# B&R Automation Studio project Nitto (part 10)

#### FB_AxisCrtl_Home.st
```iecst
(********************************************************************
 * COPYRIGHT -- Microsoft
 ********************************************************************
 * Library: Bibliothek
 * Datei: FB_AxisCrtl_Home.st
 * Autor: awalz
 * Erstellt: 23. Juli 2014
 ********************************************************************
 * Implementierung der Library Bibliothek
 ********************************************************************)

(* TODO: Bitte Kommentar hier einfügen *)
FUNCTION_BLOCK FB_AxisCrtl_Home

(***************************************************************
        Control Sequence
***************************************************************)
(* status information is read before the step sequencer to attain a shorter reaction time *)
(************************ MC_READSTATUS *************************)
	MC_ReadStatus_0.Enable :=  NOT MC_ReadStatus_0.Error;
	MC_ReadStatus_0.Axis := AxisREF;
	MC_ReadStatus_0();
	BasicControl.AxisState.Disabled             := MC_ReadStatus_0.Disabled;
	BasicControl.AxisState.StandStill           := MC_ReadStatus_0.StandStill;
	BasicControl.AxisState.Stopping             := MC_ReadStatus_0.Stopping;
	BasicControl.AxisState.Homing               := MC_ReadStatus_0.Homing;
	BasicControl.AxisState.DiscreteMotion       := MC_ReadStatus_0.DiscreteMotion;
	BasicControl.AxisState.ContinuousMotion     := MC_ReadStatus_0.ContinuousMotion;
	BasicControl.AxisState.SynchronizedMotion   := MC_ReadStatus_0.SynchronizedMotion;
	BasicControl.AxisState.ErrorStop            := MC_ReadStatus_0.Errorstop;
	BasicControl.AxisState.Homed				:= BasicControl.Status.DriveStatus.HomingOk;
	(********************MC_BR_READDRIVESTATUS***********************)
	MC_BR_ReadDriveStatus_0.Enable := NOT(MC_BR_ReadDriveStatus_0.Error);
	MC_BR_ReadDriveStatus_0.Axis := AxisREF;
	MC_BR_ReadDriveStatus_0.AdrDriveStatus := ADR(BasicControl.Status.DriveStatus);
	MC_BR_ReadDriveStatus_0();

	(******************** MC_READACTUALPOSITION *********************)
	MC_ReadActualPosition_0.Enable := (NOT(MC_ReadActualPosition_0.Error));
	MC_ReadActualPosition_0.Axis := AxisREF;
	MC_ReadActualPosition_0();
	IF(MC_ReadActualPosition_0.Valid = TRUE)THEN
		BasicControl.Status.ActPosition := MC_ReadActualPosition_0.Position;
	END_IF

	(******************** MC_READACTUALVELOCITY *********************)
	MC_ReadActualVelocity_0.Enable := (NOT(MC_ReadActualVelocity_0.Error));
	MC_ReadActualVelocity_0.Axis := AxisREF;
	MC_ReadActualVelocity_0();
	IF(MC_ReadActualVelocity_0.Valid = TRUE)THEN
		BasicControl.Status.ActVelocity := MC_ReadActualVelocity_0.Velocity;
	END_IF
	(*********************+*Parameter schreiben**********************)
	MC_MoveVelocity_0.Acceleration  := ruck;
	MC_MoveVelocity_0.Deceleration  := ruck;
	MC_ReadStatus_0();
	(************************ MC_READAXISERROR **********************)
	MC_ReadAxisError_0.Enable := NOT(MC_ReadAxisError_0.Error);
	MC_ReadAxisError_0.Axis := AxisREF;
	MC_ReadAxisError_0.DataAddress := ADR(BasicControl.Status.ErrorText);
	MC_ReadAxisError_0.DataLength := SIZEOF(BasicControl.Status.ErrorText);
	MC_ReadAxisError_0.DataObjectName := 'acp10etxde';
	MC_ReadAxisError_0();

	MC_refSwitchConfig_0.Axis := AxisREF;
	MC_refSwitchConfig_0();

	(* central monitoring OF stop command attains a shorter reaction TIME in CASE OF emergency stop *)
	(******************CHECK FOR STOP COMMAND************************)
	(*IF (BasicControl.Command.Stop = TRUE) THEN*)
	IF cmd = CONST.AXIS.STOP THEN
		IF ((AxisStep >= STATE_READY) AND (AxisStep < STATE_ERROR)) THEN
			(* reset all FB execute inputs we use *)
			MC_Home_0.Execute := 0;
			MC_Stop_0.Execute := 0;
			MC_MoveAbsolute_0.Execute := 0;
			MC_MoveAdditive_0.Execute := 0;
			MC_MoveVelocity_0.Execute := 0;
			MC_ReadAxisError_0.Acknowledge := 0;
			MC_Reset_0.Execute := 0;

			(* reset user commands *)
			BasicControl.Command.Stop := 0;
			BasicControl.Command.Home := 0;
			BasicControl.Command.MoveJogPos := 0;
			BasicControl.Command.MoveJogNeg := 0;
			BasicControl.Command.MoveVelocity := 0;
			BasicControl.Command.MoveAbsolute := 0;
			BasicControl.Command.MoveAdditive := 0;
			AxisStep := STATE_STOP;
		END_IF
	END_IF

//////////////////////////////////////////////////////////////////////////
(*	IF AxisHandle[tempIndex].AxisState.Stopping THEN
	    IF (AxisHandle[tempIndex].Status.ActVelocity = 0.0) THEN
			AxisIf.Status.isMoving 						:= FALSE;
			AllDrives.Status.stopActive					:= FALSE;
		ELSE
			AxisIf.Status.isMoving 						:= TRUE;
		END_IF
	ELSIF (NOT ( AxisHandle[tempIndex].AxisState.DiscreteMotion OR
	             AxisHandle[tempIndex].AxisState.ContinuousMotion)) THEN
		AxisIf.Status.isMoving 							:= FALSE;
		AllDrives.Status.stopActive						:= FALSE;
	ELSE
		AxisIf.Status.isMoving 							:= TRUE;
	END_IF*)
////////////////////////////////////////////////////////////////////////////
	(**************** CHECK FOR GENERAL AXIS ERROR ******************)
(*	IF ((MC_ReadAxisError_0.AxisErrorID <> 0) AND (MC_ReadAxisError_0.Valid)) THEN
		AxisStep := STATE_ERROR_AXIS;
		(***************** CHECK IF POWER SHOULD BE OFF *******************)
(*	ELSIF ((NOT BasicControl.Command.Power) AND (MC_ReadAxisError_0.Valid)) THEN
		IF ((MC_ReadStatus_0.Errorstop) AND (MC_ReadStatus_0.Valid )) THEN
			AxisStep := STATE_ERROR_RESET;
		ELSE
			AxisStep := STATE_WAIT;
		END_IF
	END_IF*)

	CASE AxisStep OF

//		******************* WAIT ************************
		STATE_WAIT:  (* STATE: Wait *)
			AxisStep := STATE_QUIT;
//			(*IF (BasicControl.Command.Power = TRUE) THEN*)
//			IF cmd = CONST.AXIS.POWER_ON THEN
//				cmdtmp := cmd;
//				AxisStep := STATE_POWER_ON;
//			ELSIF cmd = CONST.AXIS.VAXIS_ON THEN
//				cmdtmp := cmd;
//				AxisStep := STATE_VAXIS_ON;
//			ELSIF cmd = CONST.AXIS.POWER_OFF THEN
//				cmdtmp := cmd;
//				AxisStep := STATE_POWER_OFF;
//			ELSE
//				MC_Power_0.Enable := FALSE;
//			END_IF
//
//			(* reset all FB execute inputs we use *)
//			MC_Home_0.Execute := FALSE;
//			MC_Stop_0.Execute := FALSE;
//			MC_MoveAbsolute_0.Execute := FALSE;
//			MC_MoveAdditive_0.Execute := FALSE;
//			MC_MoveVelocity_0.Execute := FALSE;
//			MC_ReadAxisError_0.Acknowledge := FALSE;
//			MC_Reset_0.Execute := FALSE;
//			(* reset user commands *)
//			BasicControl.Command.Stop := FALSE;
//			BasicControl.Command.Home := FALSE;
//			BasicControl.Command.MoveJogPos := FALSE;
//			BasicControl.Command.MoveJogNeg := FALSE;
//			BasicControl.Command.MoveVelocity := FALSE;
//			BasicControl.Command.MoveAbsolute := FALSE;
//			BasicControl.Command.MoveAdditive := FALSE;
//
//			BasicControl.Status.ErrorID := 0;
//		(********************Virtuelle Achse einschalten****)
		STATE_VAXIS_ON:

			IF MC_BR_ReadDriveStatus_0.Valid THEN
				cmdtmp := cmd;
				AxisStep := STATE_QUIT;
			END_IF
		(******************** POWER ON **********************)
		STATE_POWER_ON:  (* STATE: Power on *)
			(*MC_Power_0.Enable := TRUE;*)
			IF (*BasicControl.Status.DriveStatus.ControllerReady AND *) BasicControl.Status.DriveStatus.NetworkInit AND
			cmd = CONST.AXIS.POWER_ON AND NOT MC_Power_0.Status AND NOT MC_Power_0.Error THEN
				MC_Power_0.Enable := TRUE; (*erster Anlauf*)
			ELSIF MC_Power_0.Error AND cmd = CONST.AXIS.POWER_ON THEN
					MC_Power_0.Enable := FALSE ;(* if a power error occured go to error state *)
					cmdtmp := cmd;
					AxisStep := STATE_ERROR_RESET;
			ELSIF 	MC_Power_0.Status AND NOT MC_Power_0.Error THEN
					cmdtmp := cmd;
					AxisStep := STATE_QUIT;
			ELSIF MC_ReadStatus_0.Errorstop AND cmdtmp <> cmd THEN
					BasicControl.Status.ErrorID := MC_Power_0.ErrorID;
					AxisStep := STATE_ERROR;
			END_IF
		(******************** POWER OFF **********************)
		STATE_POWER_OFF:  (* STATE: Power on *)
			MC_Power_0.Enable := FALSE;
			IF NOT MC_Power_0.Status THEN
				cmdtmp := cmd;
				AxisStep := STATE_QUIT;
			END_IF
			(* if a power error occured go to error state *)
			IF MC_Power_0.Error  THEN
				BasicControl.Status.ErrorID := MC_Power_0.ErrorID;
				AxisStep := STATE_ERROR;
			ELSIF MC_ReadStatus_0.Errorstop AND cmdtmp <> cmd THEN
				AxisStep := STATE_ERROR_RESET;
			END_IF
		(******************** READY **********************)
		STATE_READY:  (* STATE: Waiting for commands *)
			IF cmd <> CONST.AXIS.NOACTION THEN
					busy := TRUE;
					cmdtmp:= cmd;
					IF cmd = CONST.AXIS.RESET THEN
						AxisStep := STATE_ERROR_RESET;
					ELSIF cmd = CONST.AXIS.STOP THEN
						MC_Stop_0( Execute := TRUE, Deceleration := verzoegerung);
						AxisStep := STATE_STOP;
					ELSIF cmd = CONST.AXIS.JOG_NEG THEN
						MC_MoveVelocity_0(Execute := TRUE, Velocity := 16666*velocity,Direction := mcNEGATIVE_DIR,
								Acceleration  := BasicControl.Parameter.Acceleration, Deceleration := BasicControl.Parameter.Deceleration);
						AxisStep := STATE_JOG_NEGATIVE;
					ELSIF cmd = CONST.AXIS.JOG_POS THEN
						MC_MoveVelocity_0(Execute := TRUE, Velocity := 16666*velocity,Direction := mcPOSITIVE_DIR,
									Acceleration  := BasicControl.Parameter.Acceleration, Deceleration := BasicControl.Parameter.Deceleration);
						AxisStep := STATE_JOG_POSITIVE;
					ELSIF cmd = CONST.AXIS.SETPOS THEN
						MC_MoveAbsolute_0(Execute := TRUE, Position := position, Velocity := 16666*velocity, Direction := mcPOSITIVE_DIR,
								Acceleration  := BasicControl.Parameter.Acceleration, Deceleration := BasicControl.Parameter.Deceleration);
						AxisStep := STATE_MOVE_ABSOLUTE; (*STATE_MOVE_ADDITIVE*)(*STATE_MOVE_ABSOLUTE;*)
					ELSIF  cmd = CONST.AXIS.CALIBR THEN
						MC_Home_0(Execute := TRUE, Position := BasicControl.Parameter.HomePosition, HomingMode := BasicControl.Parameter.HomeMode);
						AxisStep := STATE_HOME;
					ELSIF cmd = CONST.AXIS.MOVE_VELOCITY THEN
							MC_MoveVelocity_0(Execute := TRUE, Velocity := 16666*velocity,Direction := mcPOSITIVE_DIR);
						AxisStep := STATE_MOVE_VELOCITY;
					ELSIF   cmd = CONST.AXIS.POWER_OFF THEN
						AxisStep := STATE_POWER_OFF;
					ELSIF   cmd = CONST.AXIS.POWER_ON THEN
						AxisStep := STATE_POWER_ON;
					END_IF
			(*ELSE
				busy := FALSE;*)
			END_IF
		(******************** HOME **********************)
		STATE_HOME:  (* STATE: start homing process *)
//			IF cmd = CONST.AXIS.CALIBR AND NOT MC_Home_0.Done THEN
//				MC_Home_0.Execute := TRUE;
			IF MC_Home_0.Done AND cmd = CONST.AXIS.CALIBR THEN
				MC_Home_0.Execute := FALSE;
				BasicControl.AxisState.Homed := TRUE;
				cmdtmp := cmd;
				busy := FALSE;
				AxisStep := STATE_QUIT;
			ELSIF cmd <> CONST.AXIS.CALIBR THEN
				MC_Home_0.Execute := FALSE;
				MC_Stop_0( Execute := TRUE, Deceleration := verzoegerung);
				AxisStep := STATE_STOP;
			END_IF
			(* if a homing error occured go to error state *)
			IF MC_Home_0.Error  OR MC_ReadStatus_0.Errorstop THEN
				MC_Home_0.Execute := FALSE;
				BasicControl.Status.ErrorID := MC_Home_0.ErrorID;
				AxisStep := STATE_ERROR;
			END_IF

		(***********************HALT_MOVEMENT***************************)
		STATE_HALT:   (* STATE: Halt movement *)
			MC_Halt_0.Deceleration := BasicControl.Parameter.Deceleration;
			MC_Halt_0.Execute := TRUE;
			IF MC_Halt_0.Done OR MC_Halt_0.CommandAborted THEN
				MC_Halt_0.Execute := FALSE;
				cmdtmp := cmd;
				busy := FALSE;
				AxisStep := STATE_QUIT;
			ELSIF cmd = CONST.AXIS.STOP THEN
				MC_Halt_0.Execute := FALSE;
				MC_Stop_0( Execute := TRUE, Deceleration := verzoegerung);
				AxisStep := STATE_STOP;
			END_IF
			(* check if error occured *)
			IF MC_Halt_0.Error OR  MC_ReadStatus_0.Errorstop THEN
				BasicControl.Status.ErrorID := MC_Halt_0.ErrorID;
				MC_Halt_0.Execute := FALSE;
				AxisStep := STATE_ERROR;
			END_IF

		(*********************** STOP MOVEMENT *************************)
		STATE_STOP: //9  (* STATE: Stop movement *)
			(* if axis is stopped go to ready state *)
			MC_Stop_0.Execute := TRUE;
			IF MC_Stop_0.Done OR MC_ReadStatus_0.StandStill THEN
				MC_Stop_0.Execute := FALSE;
				cmdtmp := cmd;
				AxisStep := STATE_QUIT;
			ELSIF MC_ReadStatus_0.Disabled THEN
				MC_Stop_0.Execute := FALSE;
				cmdtmp := cmd;
				AxisStep := STATE_QUIT;
			END_IF
			(* check if error occured *)
			IF MC_Stop_0.Error OR MC_ReadStatus_0.Errorstop THEN
				BasicControl.Status.ErrorID := MC_Stop_0.ErrorID;
				MC_Stop_0.Execute := FALSE;
				AxisStep := STATE_ERROR;
			END_IF

		(******************** START JOG MOVEMENT POSITVE **********************)
		STATE_JOG_POSITIVE:  (* STATE: Start jog movement in positive direction *)
			IF cmd <> CONST.AXIS.JOG_POS AND cmd <> CONST.AXIS.STOP THEN
				cmdtmp := cmd;
				MC_MoveVelocity_0.Execute := FALSE;
				AxisStep := STATE_HALT;
			ELSIF cmd = CONST.AXIS.STOP THEN
				MC_MoveVelocity_0.Execute := FALSE;
				MC_Stop_0( Execute := TRUE, Deceleration := verzoegerung);
				AxisStep := STATE_STOP;
			END_IF
			(* check if error occured *)
			IF MC_MoveVelocity_0.Error OR MC_ReadStatus_0.Errorstop  THEN
				BasicControl.Status.ErrorID := MC_MoveVelocity_0.ErrorID;
				MC_MoveVelocity_0.Execute := FALSE;
				AxisStep := STATE_ERROR;
			END_IF

		(******************** START JOG MOVEMENT NEGATIVE **********************)
		STATE_JOG_NEGATIVE:  (* STATE: Start jog movement in negative direction *)

			IF cmd <> CONST.AXIS.JOG_NEG AND  cmd <> CONST.AXIS.STOP THEN
				MC_MoveVelocity_0.Execute := FALSE;
				cmdtmp := cmd;
				AxisStep := STATE_HALT;
			ELSIF cmd = CONST.AXIS.STOP THEN
				MC_MoveVelocity_0.Execute := FALSE;
				MC_Stop_0( Execute := TRUE, Deceleration := verzoegerung);
				AxisStep := STATE_STOP;
			END_IF
			(* check if error occured *)
			IF MC_MoveVelocity_0.Error OR MC_ReadStatus_0.Errorstop THEN
				BasicControl.Status.ErrorID := MC_MoveVelocity_0.ErrorID;
				MC_MoveVelocity_0.Execute := FALSE;
				AxisStep := STATE_ERROR;
			END_IF

		(******************** START ABSOLUTE MOVEMENT **********************)
		STATE_MOVE_ABSOLUTE:  (* STATE: Start absolute movement *)
			(* check if commanded position is reached *)
			IF cmd <> CONST.AXIS.SETPOS AND cmd <> CONST.AXIS.STOP  THEN
				MC_MoveAbsolute_0.Execute := FALSE;
				cmdtmp := cmd;
				AxisStep := STATE_HALT;
			ELSIF MC_MoveAbsolute_0.Done THEN
				MC_MoveAbsolute_0.Execute := FALSE;
				cmdtmp := cmd;
				AxisStep := STATE_QUIT;
			ELSIF cmd = CONST.AXIS.STOP THEN
				MC_MoveAbsolute_0.Execute := FALSE;
				MC_Stop_0.Deceleration := verzoegerung;
				MC_Stop_0.Execute := TRUE;
				AxisStep := STATE_STOP;
			END_IF
			(* check if error occured *)
			IF MC_MoveAbsolute_0.Error OR MC_ReadStatus_0.Errorstop THEN
				BasicControl.Status.ErrorID := MC_MoveAbsolute_0.ErrorID;
				MC_MoveAbsolute_0.Execute := TRUE;
				AxisStep := STATE_ERROR;
			END_IF

		(******************** START ADDITIVE MOVEMENT **********************)
		STATE_MOVE_ADDITIVE:  (* STATE: Start additive movement *)
			(*	MC_MoveAdditive_0.Distance      := BasicControl.Parameter.Distance;
			MC_MoveAdditive_0.Velocity      := BasicControl.Parameter.Velocity;
			MC_MoveAdditive_0.Execute := TRUE;*)
			MC_MoveAdditive_0.Acceleration  := BasicControl.Parameter.Acceleration;
			MC_MoveAdditive_0.Deceleration  := BasicControl.Parameter.Deceleration;

			(* check if commanded distance is reached *)
			IF cmd <> CONST.AXIS.SETPOS AND cmd <> CONST.AXIS.STOP THEN
				MC_MoveAdditive_0.Execute := FALSE;
				cmdtmp := cmd;
				AxisStep := STATE_HALT;
			ELSIF MC_MoveAdditive_0.Done  THEN
				MC_MoveAdditive_0.Execute := FALSE;
				cmdtmp := cmd;
				AxisStep := STATE_QUIT;
			ELSIF cmd = CONST.AXIS.STOP THEN
				MC_MoveAdditive_0.Execute := FALSE;
				MC_Stop_0( Execute := TRUE, Deceleration := verzoegerung);
				AxisStep := STATE_STOP;
			END_IF
			(* check if error occured *)
			IF MC_MoveAdditive_0.Error OR  MC_ReadStatus_0.Errorstop THEN
				BasicControl.Status.ErrorID := MC_MoveAdditive_0.ErrorID;
				MC_MoveAdditive_0.Execute := FALSE;
				AxisStep := STATE_ERROR;
			END_IF

		(******************** START VELOCITY MOVEMENT **********************)
		STATE_MOVE_VELOCITY:  (* STATE: Start velocity movement *)
					(* check if commanded velocity is reached *)
			IF cmd <>  CONST.AXIS.MOVE_VELOCITY AND  cmd <> CONST.AXIS.STOP THEN
				MC_MoveVelocity_0.Execute := FALSE;
				cmdtmp := cmd;
				AxisStep := STATE_HALT;
			ELSIF MC_MoveVelocity_0.InVelocity THEN
				MC_MoveVelocity_0.Execute := FALSE;
				cmdtmp := cmd;
				AxisStep := STATE_QUIT;
			ELSIF cmd = CONST.AXIS.STOP THEN
				MC_MoveVelocity_0.Execute := FALSE;
				MC_Stop_0( Execute := TRUE, Deceleration := verzoegerung);
				AxisStep := STATE_STOP;
			END_IF
			(* check if error occured *)
			IF MC_MoveVelocity_0.Error OR MC_ReadStatus_0.Errorstop THEN
				BasicControl.Status.ErrorID := MC_MoveVelocity_0.ErrorID;
				MC_MoveVelocity_0.Execute := FALSE;
				AxisStep := STATE_ERROR;
			END_IF

		(******************** FB-ERROR OCCURED *************************)
		STATE_ERROR:  (* STATE: Error *)
			(* check if FB indicates an axis error *)
			IF (MC_ReadAxisError_0.AxisErrorCount<>0) THEN
				AxisStep := STATE_ERROR_AXIS;
			ELSE
				IF (BasicControl.Command.ErrorAcknowledge = TRUE) THEN
					BasicControl.Command.ErrorAcknowledge := FALSE;
					BasicControl.Status.ErrorID := 0;
					(* reset axis if it is in axis state ErrorStop *)
					IF MC_ReadStatus_0.Errorstop AND MC_ReadStatus_0.Valid  THEN
						AxisStep := STATE_ERROR_RESET;
					ELSE
						cmdtmp := cmd;
						AxisStep := STATE_QUIT;
					END_IF
				END_IF
			END_IF

		(******************** AXIS-ERROR OCCURED *************************)
		STATE_ERROR_AXIS:  (* STATE: Axis Error *)
			IF (MC_ReadAxisError_0.Valid) THEN
			err.set := TRUE;
			err.text := MC_ReadAxisError_0.DataObjectName;
			err.id :=  UINT_TO_DINT  (MC_ReadAxisError_0.AxisErrorID) ;
				IF (MC_ReadAxisError_0.AxisErrorID <> 0) THEN
					BasicControl.Status.ErrorID := MC_ReadAxisError_0.AxisErrorID;
				END_IF
				MC_ReadAxisError_0.Acknowledge := FALSE;
			(*	IF (BasicControl.Command.ErrorAcknowledge) THEN
					BasicControl.Command.ErrorAcknowledge := FALSE;
					(* acknowledge axis error *)
				IF cmd = CONST.AXIS.RESET THEN
					IF (MC_ReadAxisError_0.AxisErrorID <> 0) THEN
						MC_ReadAxisError_0.Acknowledge := TRUE;
						AxisStep := STATE_ERROR_RESET;
					END_IF
				END_IF
				IF (MC_ReadAxisError_0.AxisErrorCount = 0) THEN
					(* reset axis if it is in axis state ErrorStop *)
					BasicControl.Status.ErrorID := 0;
					IF ((MC_ReadStatus_0.Errorstop ) AND (MC_ReadStatus_0.Valid)) THEN
						AxisStep := STATE_ERROR_RESET;
					ELSE
						(*AxisStep := STATE_WAIT;*)
						cmdtmp := cmd;
						AxisStep := STATE_QUIT;
					END_IF
				ELSIF NOT MC_ReadAxisError_0.Error THEN
						cmdtmp := cmd;
							AxisStep := STATE_QUIT;
				END_IF
			ELSE
				AxisStep := STATE_WAIT; (* kein Fehler liegt vor*)
			END_IF

		(******************** RESET DONE *************************)
		STATE_ERROR_RESET:  (* STATE: Wait for reset done *)
			MC_Reset_0.Execute := TRUE;
			(* reset MC_Power.Enable if this FB is in Error*)
			IF (MC_Power_0.Error) THEN
				MC_Power_0.Enable := FALSE;
			END_IF
			IF(MC_Reset_0.Done)THEN
				MC_Reset_0.Execute := FALSE;
				(*AxisStep := STATE_WAIT;*)
				cmdtmp := cmd;
				(*cmd := CONST.AXIS.NOACTION;*)
				AxisStep := STATE_QUIT;
			ELSIF(MC_Reset_0.Error) THEN
				MC_Reset_0.Execute := FALSE;
				AxisStep := STATE_ERROR;
			END_IF
			(******************** SEQUENCE END *************************)
		STATE_QUIT:
		(*IF cmd = CONST.CUTTINGUNIT.CMDs.ABORT THEN
			busy := TRUE;
			state := ST_ABORT;
		ELSE*)
			busy := FALSE;
			IF cmd = cmdtmp THEN
				busy := FALSE;
				cmd := CONST.AXIS.NOACTION;
				AxisStep := STATE_READY;
			ELSIF cmd <> CONST.AXIS.NOACTION THEN
				busy := FALSE;
				AxisStep := STATE_READY;
			(*ELSIF cmd = CONST.AXIS.POWER_OFF THEN
				cmdtmp := cmd;
				AxisStep := STATE_POWER_OFF;*)
			(*ELSIF cmd = CONST.AXIS.POWER_ON THEN
				cmdtmp := cmd;
				AxisStep := STATE_POWER_ON;*)

			END_IF

	END_CASE

(***************************************************************
        FUNCTION Block Calls
***************************************************************)

(************************** MC_POWER ****************************)
	MC_Power_0.Axis := AxisREF;  (* pointer to axis *)
	MC_Power_0();

	(************************** MC_HOME *****************************)
	MC_Home_0.Axis := AxisREF;
	MC_Home_0();

	(********************** MC_MOVEABSOLUTE *************************)
	MC_MoveAbsolute_0.Axis := AxisREF;
	MC_MoveAbsolute_0();

	(********************** MC_MOVEADDITIVE *************************)
	MC_MoveAdditive_0.Axis := AxisREF;
	MC_MoveAdditive_0();

	(********************** MC_MOVEVELOCITY *************************)
	MC_MoveVelocity_0.Axis := AxisREF;
	MC_MoveVelocity_0();

	(************************** MC_STOP *****************************)
	MC_Stop_0.Axis := AxisREF;
	MC_Stop_0();

	(***************************MC_HALT******************************)
	MC_Halt_0.Axis := AxisREF;
	MC_Halt_0();

	(************************** MC_RESET ****************************)
	MC_Reset_0.Axis := AxisREF;
	MC_Reset_0();
END_FUNCTION_BLOCK
```

#### FB_AxisState.st
```iecst
(********************************************************************
 * COPYRIGHT -- Microsoft
 ********************************************************************
 * Library: Bibliothek
 * Datei: FB_AxisState.st
 * Autor: awalz
 * Erstellt: 26. August 2014
 ********************************************************************
 * Implementierung der Library Bibliothek
 ********************************************************************)

(* TODO: Bitte Kommentar hier einfügen *)
FUNCTION_BLOCK FB_AxisState
//		Error:				INT:=1;
//		Errorstop:			INT:=2;
//		Disabled:			INT:=3;
//		Stopping:			INT:=4;
//		StandStill:			INT:=5;
//		DiscreteMotion:		INT:=6;
//		ContinuousMotion: 	INT:=7;
//		SynchronizedMotion:	INT:=8;
//		Homing:				INT:=9;
	stati[CONST.Error] := readstatus.Error;
	stati[CONST.Errorstop] :=	readstatus.Errorstop;
	stati[CONST.Disabled] :=	readstatus.Disabled;
	stati[3] :=	readstatus.Stopping;
	stati[4] := readstatus.StandStill;
	stati[5] := readstatus.DiscreteMotion;
	stati[6] :=	readstatus.ContinuousMotion;
	stati[7] :=	readstatus.SynchronizedMotion;
//	CONST.texts[CONST.Error] := stati[0];
//
//
//		readstatus.SynchronizedMotion
END_FUNCTION_BLOCK
```

#### FB_AxisCtrl_GridFeeder.st
```iecst
(********************************************************************
 * COPYRIGHT -- Microsoft
 ********************************************************************
 * Library: Bibliothek
 * Datei: FB_AxisCtrl.st
 * Autor: awalz
 * Erstellt: 23. Juli 2014
 ********************************************************************
 * Implementierung der Library Bibliothek
 ********************************************************************)

(* TODO: Bitte Kommentar hier einfügen *)
FUNCTION_BLOCK FB_AxisCtrl_GridFeeder

(***************************************************************
        Control Sequence
***************************************************************)
(* status information is read before the step sequencer to attain a shorter reaction time *)
(************************ MC_READSTATUS *************************)
	MC_ReadStatus_0.Enable :=  NOT MC_ReadStatus_0.Error;
	MC_ReadStatus_0.Axis := AxisREF;
	MC_ReadStatus_0();
	BasicControl.AxisState.Disabled             := MC_ReadStatus_0.Disabled;
	BasicControl.AxisState.StandStill           := MC_ReadStatus_0.StandStill;
	BasicControl.AxisState.Stopping             := MC_ReadStatus_0.Stopping;
	BasicControl.AxisState.Homing               := MC_ReadStatus_0.Homing;
	BasicControl.AxisState.DiscreteMotion       := MC_ReadStatus_0.DiscreteMotion;
	BasicControl.AxisState.ContinuousMotion     := MC_ReadStatus_0.ContinuousMotion;
	BasicControl.AxisState.SynchronizedMotion   := MC_ReadStatus_0.SynchronizedMotion;
	BasicControl.AxisState.ErrorStop            := MC_ReadStatus_0.Errorstop;

	(********************MC_BR_READDRIVESTATUS***********************)
	MC_BR_ReadDriveStatus_0.Enable := NOT(MC_BR_ReadDriveStatus_0.Error);
	MC_BR_ReadDriveStatus_0.Axis := AxisREF;
	MC_BR_ReadDriveStatus_0.AdrDriveStatus := ADR(BasicControl.Status.DriveStatus);
	MC_BR_ReadDriveStatus_0();

	(******************** MC_READACTUALPOSITION *********************)
	MC_ReadActualPosition_0.Enable := (NOT(MC_ReadActualPosition_0.Error));
	MC_ReadActualPosition_0.Axis := AxisREF;
	MC_ReadActualPosition_0();
	IF(MC_ReadActualPosition_0.Valid = TRUE)THEN
		BasicControl.Status.ActPosition := MC_ReadActualPosition_0.Position;
	END_IF

	(******************** MC_READACTUALVELOCITY *********************)
	MC_ReadActualVelocity_0.Enable := (NOT(MC_ReadActualVelocity_0.Error));
	MC_ReadActualVelocity_0.Axis := AxisREF;
	MC_ReadActualVelocity_0();
	IF(MC_ReadActualVelocity_0.Valid = TRUE)THEN
		BasicControl.Status.ActVelocity := MC_ReadActualVelocity_0.Velocity;
	END_IF
	(*********************+*Parameter schreiben**********************)
	MC_MoveVelocity_0.Acceleration  := ruck;
	MC_MoveVelocity_0.Deceleration  := ruck;
	MC_ReadStatus_0();
	(************************ MC_READAXISERROR **********************)
	MC_ReadAxisError_0.Enable := NOT(MC_ReadAxisError_0.Error);
	MC_ReadAxisError_0.Axis := AxisREF;
	MC_ReadAxisError_0.DataAddress := ADR(BasicControl.Status.ErrorText);
	MC_ReadAxisError_0.DataLength := SIZEOF(BasicControl.Status.ErrorText);
	MC_ReadAxisError_0.DataObjectName := 'acp10etxde';
	MC_ReadAxisError_0();
	(* central monitoring OF stop command attains a shorter reaction TIME in CASE OF emergency stop *)
	(******************CHECK FOR STOP COMMAND************************)
	(*IF (BasicControl.Command.Stop = TRUE) THEN*)
	//	IF cmd = CONST.AXIS.STOP THEN //12.03.15
	//		busy := TRUE;
	//		IF ((AxisStep >= STATE_READY) AND (AxisStep < STATE_ERROR)) THEN
	//			(* reset all FB execute inputs we use *)
	//			MC_Home_0.Execute := 0;
	//			MC_Stop_0.Execute := 0;
	//			MC_MoveAbsolute_0.Execute := 0;
	//			MC_MoveAdditive_0.Execute := 0;
	//			MC_MoveVelocity_0.Execute := 0;
	//			MC_ReadAxisError_0.Acknowledge := 0;
	//			MC_Reset_0.Execute := 0;
	//
	//			(* reset user commands *)
	//			BasicControl.Command.Stop := 0;
	//			BasicControl.Command.Home := 0;
	//			BasicControl.Command.MoveJogPos := 0;
	//			BasicControl.Command.MoveJogNeg := 0;
	//			BasicControl.Command.MoveVelocity := 0;
	//			BasicControl.Command.MoveAbsolute := 0;
	//			BasicControl.Command.MoveAdditive := 0;
	//			MC_Stop_0( Execute := TRUE, Deceleration := verzoegerung);
	//			AxisStep := STATE_STOP;
	//		END_IF
	//	END_IF
	//
	////////////////////////////////////////////////////////////////////////////
	//(*	IF AxisHandle[tempIndex].AxisState.Stopping THEN
	//	    IF (AxisHandle[tempIndex].Status.ActVelocity = 0.0) THEN
	//			AxisIf.Status.isMoving 						:= FALSE;
	//			AllDrives.Status.stopActive					:= FALSE;
	//		ELSE
	//			AxisIf.Status.isMoving 						:= TRUE;
	//		END_IF
	//	ELSIF (NOT ( AxisHandle[tempIndex].AxisState.DiscreteMotion OR
	//	             AxisHandle[tempIndex].AxisState.ContinuousMotion)) THEN
	//		AxisIf.Status.isMoving 							:= FALSE;
	//		AllDrives.Status.stopActive						:= FALSE;
	//	ELSE
	//		AxisIf.Status.isMoving 							:= TRUE;
	//	END_IF*)
	//////////////////////////////////////////////////////////////////////////////
	//	(**************** CHECK FOR GENERAL AXIS ERROR ******************)
	//(*	IF ((MC_ReadAxisError_0.AxisErrorID <> 0) AND (MC_ReadAxisError_0.Valid)) THEN
	//		AxisStep := STATE_ERROR_AXIS;
	//		(***************** CHECK IF POWER SHOULD BE OFF *******************)
	//(*	ELSIF ((NOT BasicControl.Command.Power) AND (MC_ReadAxisError_0.Valid)) THEN
	//		IF ((MC_ReadStatus_0.Errorstop) AND (MC_ReadStatus_0.Valid )) THEN
	//			AxisStep := STATE_ERROR_RESET;
	//		ELSE
	//			AxisStep := STATE_WAIT;
	//		END_IF
	//	END_IF*)

	CASE AxisStep OF

		//		******************* WAIT ************************
		STATE_WAIT:  (* STATE: Wait *)
			AxisStep := STATE_QUIT;
		//			(*IF (BasicControl.Command.Power = TRUE) THEN*)
		//			IF cmd = CONST.AXIS.POWER_ON THEN
		//				cmdtmp := cmd;
		//				AxisStep := STATE_POWER_ON;
		//			ELSIF cmd = CONST.AXIS.VAXIS_ON THEN
		//				cmdtmp := cmd;
		//				AxisStep := STATE_VAXIS_ON;
		//			ELSIF cmd = CONST.AXIS.POWER_OFF THEN
		//				cmdtmp := cmd;
		//				AxisStep := STATE_POWER_OFF;
		//			ELSE
		//				MC_Power_0.Enable := FALSE;
		//			END_IF
		//
		//			(* reset all FB execute inputs we use *)
		//			MC_Home_0.Execute := FALSE;
		//			MC_Stop_0.Execute := FALSE;
		//			MC_MoveAbsolute_0.Execute := FALSE;
		//			MC_MoveAdditive_0.Execute := FALSE;
		//			MC_MoveVelocity_0.Execute := FALSE;
		//			MC_ReadAxisError_0.Acknowledge := FALSE;
		//			MC_Reset_0.Execute := FALSE;
		//			(* reset user commands *)
		//			BasicControl.Command.Stop := FALSE;
		//			BasicControl.Command.Home := FALSE;
		//			BasicControl.Command.MoveJogPos := FALSE;
		//			BasicControl.Command.MoveJogNeg := FALSE;
		//			BasicControl.Command.MoveVelocity := FALSE;
		//			BasicControl.Command.MoveAbsolute := FALSE;
		//			BasicControl.Command.MoveAdditive := FALSE;
		//
		//			BasicControl.Status.ErrorID := 0;
		//		(********************Virtuelle Achse einschalten****)
		STATE_VAXIS_ON:

			IF MC_BR_ReadDriveStatus_0.Valid THEN
				cmdtmp := cmd;
				AxisStep := STATE_QUIT;
			END_IF
		(******************** POWER ON **********************)
		STATE_POWER_ON:  (* STATE: Power on *)
			(*MC_Power_0.Enable := TRUE;*)
			IF BasicControl.Status.DriveStatus.ControllerReady AND	cmd = CONST.AXIS.POWER_ON
				AND NOT MC_Power_0.Status AND NOT MC_Power_0.Error THEN
				MC_Power_0.Enable := TRUE; (*erster Anlauf*)
				cmdtmp := cmd;
			ELSIF MC_Power_0.Error AND cmdtmp = cmd THEN
				MC_Power_0.Enable := FALSE ;(* if a power error occured go to error state *)
				cmd := CONST.AXIS.RESET;
				AxisStep := STATE_ERROR_RESET;
			ELSIF 	MC_Power_0.Status AND NOT MC_Power_0.Error THEN
				cmdtmp := cmd;
				AxisStep := STATE_QUIT;
		(*	ELSIF MC_Power_0.Error AND cmdtmp <> cmd THEN
					BasicControl.Status.ErrorID := MC_Power_0.ErrorID;
					AxisStep := STATE_ERROR;*)
			ELSIF MC_ReadStatus_0.Errorstop THEN (*24.07.14*)
				BasicControl.Status.ErrorID := MC_Power_0.ErrorID;
				cmdtmp := cmd;
				AxisStep := STATE_ERROR;
			END_IF
		(******************** POWER OFF **********************)
		STATE_POWER_OFF:  (* STATE: Power on *)
			MC_Power_0.Enable := FALSE;
			IF NOT MC_Power_0.Status THEN
				cmdtmp := cmd;
				(*AxisStep := STATE_READY;*)
				AxisStep := STATE_QUIT;
			END_IF
			(* if a power error occured go to error state *)
			IF MC_Power_0.Error  THEN
				BasicControl.Status.ErrorID := MC_Power_0.ErrorID;
				AxisStep := STATE_ERROR;
			END_IF
		(******************** READY **********************)
		STATE_READY:  (* STATE: Waiting for commands *)
			IF cmd <> CONST.AXIS.NOACTION THEN
				busy := TRUE;
				(*cmdtmp:= cmd; *)//13.03.15
				IF cmd = CONST.AXIS.RESET THEN
					AxisStep := STATE_ERROR_RESET;
				ELSIF cmd = CONST.AXIS.STOP THEN
					MC_Stop_0( Execute := TRUE, Deceleration := verzoegerung);
					AxisStep := STATE_STOP;
				ELSIF cmd = CONST.AXIS.JOG_NEG THEN
					MC_MoveVelocity_0(Execute := TRUE, Velocity := 16666*velocity, Acceleration := BasicControl.Parameter.Acceleration,
					Deceleration  := BasicControl.Parameter.Deceleration, Direction := mcNEGATIVE_DIR);
					AxisStep := STATE_JOG_NEGATIVE;
				ELSIF cmd = CONST.AXIS.JOG_POS THEN
					MC_MoveVelocity_0(Execute := TRUE, Velocity := 16666*velocity, Acceleration := BasicControl.Parameter.Acceleration,
					Deceleration  := BasicControl.Parameter.Deceleration,Direction := mcPOSITIVE_DIR);
					AxisStep := STATE_JOG_POSITIVE;
				ELSIF cmd = CONST.AXIS.SETPOS THEN
					MC_MoveAbsolute_0(Execute := TRUE, Position := position, Velocity := 16666*velocity, Acceleration := BasicControl.Parameter.Acceleration,
					Deceleration  := BasicControl.Parameter.Deceleration, Direction := mcPOSITIVE_DIR);
					AxisStep := STATE_MOVE_ABSOLUTE;
				ELSIF  cmd = CONST.AXIS.CALIBR THEN
					(*Achse referenzieren*)
					AxisStep := STATE_HOME;
				ELSIF cmd = CONST.AXIS.MOVE_VELOCITY THEN
					//							MC_MoveVelocity_0.Acceleration  := BasicControl.Parameter.Acceleration;
					//							MC_MoveVelocity_0.Deceleration  := BasicControl.Parameter.Deceleration;
					MC_MoveVelocity_0(Execute := TRUE, Velocity := 16666*velocity, Acceleration := BasicControl.Parameter.Acceleration,
					Deceleration  := BasicControl.Parameter.Deceleration,	Direction := mcPOSITIVE_DIR);
					AxisStep := STATE_MOVE_VELOCITY;
				ELSIF   cmd = CONST.AXIS.POWER_OFF THEN
					AxisStep := STATE_POWER_OFF;
				ELSIF   cmd = CONST.AXIS.POWER_ON THEN
					AxisStep := STATE_POWER_ON;
				END_IF
			ELSE
				busy := FALSE;
			END_IF
		(******************** HOME **********************)
		STATE_HOME:  (* STATE: start homing process *)
			MC_Home_0.Position := BasicControl.Parameter.HomePosition;
			MC_Home_0.HomingMode := BasicControl.Parameter.HomeMode;
			MC_Home_0.Execute := TRUE;
			IF MC_Home_0.Done AND cmd = CONST.AXIS.CALIBR THEN
				MC_Home_0.Execute := FALSE;
				BasicControl.AxisState.Homed := TRUE;
				cmdtmp := cmd;
				AxisStep := STATE_QUIT;
			ELSIF cmd <> CONST.AXIS.CALIBR THEN
				MC_Home_0.Execute := FALSE;
				MC_Stop_0( Execute := TRUE, Deceleration := verzoegerung);
				AxisStep := STATE_STOP;
			END_IF

			(* if a homing error occured go to error state *)
			IF MC_Home_0.Error  OR MC_ReadStatus_0.Errorstop THEN
				MC_Home_0.Execute := FALSE;
				BasicControl.Status.ErrorID := MC_Home_0.ErrorID;
				AxisStep := STATE_ERROR;
			END_IF

		(***********************HALT_MOVEMENT***************************)
		STATE_HALT:   (* STATE: Halt movement *)
			MC_Halt_0.Deceleration := BasicControl.Parameter.Deceleration;
			MC_Halt_0.Execute := TRUE;
			IF MC_Halt_0.Done THEN
				MC_Halt_0.Execute := FALSE;
				cmdtmp := cmd;
				AxisStep := STATE_QUIT;
			ELSIF cmd = CONST.AXIS.STOP THEN
				MC_Halt_0.Execute := FALSE;
				MC_Stop_0( Execute := TRUE, Deceleration := verzoegerung);
				AxisStep := STATE_STOP;
			END_IF
			(* check if error occured *)
			IF MC_Halt_0.Error OR  MC_ReadStatus_0.Errorstop THEN
				BasicControl.Status.ErrorID := MC_Halt_0.ErrorID;
				MC_Halt_0.Execute := FALSE;
				AxisStep := STATE_ERROR;
			END_IF

		(*********************** STOP MOVEMENT *************************)
		STATE_STOP:  (* STATE: Stop movement *)
			//			MC_Stop_0.Deceleration := BasicControl.Parameter.Deceleration;
			//			MC_Stop_0.Execute := TRUE;
			(* if axis is stopped go to ready state *)
			IF MC_Stop_0.Done  OR MC_ReadStatus_0.StandStill THEN
				MC_Stop_0.Execute := FALSE;
				cmdtmp := cmd;
				AxisStep := STATE_QUIT;
			ELSIF MC_ReadStatus_0.Disabled THEN
				MC_Stop_0.Execute := FALSE;
				cmdtmp := cmd;
				AxisStep := STATE_QUIT;
			END_IF
			(* check if error occured *)
			IF MC_Stop_0.Error OR MC_ReadStatus_0.Errorstop THEN
				BasicControl.Status.ErrorID := MC_Stop_0.ErrorID;
				MC_Stop_0.Execute := FALSE;
				AxisStep := STATE_ERROR;
			END_IF

		(******************** START JOG MOVEMENT POSITVE **********************)
		STATE_JOG_POSITIVE:  (* STATE: Start jog movement in positive direction *)
			IF cmd <> CONST.AXIS.JOG_POS AND cmd <> CONST.AXIS.STOP THEN
				cmdtmp := cmd;
				MC_MoveVelocity_0.Execute := FALSE;
				AxisStep := STATE_HALT;
			ELSIF cmd = CONST.AXIS.STOP THEN
				MC_MoveVelocity_0.Execute := FALSE;
				MC_Stop_0( Execute := TRUE, Deceleration := verzoegerung);
				AxisStep := STATE_STOP;
			END_IF
			(* check if error occured *)
			IF MC_MoveVelocity_0.Error OR MC_ReadStatus_0.Errorstop  THEN
				BasicControl.Status.ErrorID := MC_MoveVelocity_0.ErrorID;
				MC_MoveVelocity_0.Execute := FALSE;
				AxisStep := STATE_ERROR;
			END_IF

		(******************** START JOG MOVEMENT NEGATIVE **********************)
		STATE_JOG_NEGATIVE:  (* STATE: Start jog movement in negative direction *)
			IF cmd <> CONST.AXIS.JOG_NEG AND cmd <> CONST.AXIS.STOP  THEN
				MC_MoveVelocity_0.Execute := FALSE;
				cmdtmp := cmd;
				AxisStep := STATE_HALT;
			ELSIF cmd = CONST.AXIS.STOP THEN
				MC_MoveVelocity_0.Execute := FALSE;
				MC_Stop_0( Execute := TRUE, Deceleration := verzoegerung);
				AxisStep := STATE_STOP;
			END_IF
			(* check if error occured *)
			IF MC_MoveVelocity_0.Error OR MC_ReadStatus_0.Errorstop  THEN
				BasicControl.Status.ErrorID := MC_MoveVelocity_0.ErrorID;
				MC_MoveVelocity_0.Execute := FALSE;
				AxisStep := STATE_ERROR;
			END_IF

		(******************** START ABSOLUTE MOVEMENT **********************)
		STATE_MOVE_ABSOLUTE:  (* STATE: Start absolute movement *)
			(* check if commanded position is reached *)
			IF cmd <> CONST.AXIS.SETPOS AND cmd <> CONST.AXIS.STOP THEN
				MC_MoveAbsolute_0.Execute := FALSE;
				cmdtmp := cmd;
				AxisStep := STATE_HALT;
			ELSIF MC_MoveAbsolute_0.Done  THEN
				MC_MoveAbsolute_0.Execute := FALSE;
				cmdtmp := cmd;
				AxisStep := STATE_QUIT;
			ELSIF cmd = CONST.AXIS.STOP THEN
				MC_MoveAbsolute_0.Execute := FALSE;
				MC_Stop_0( Execute := TRUE, Deceleration := verzoegerung);
				AxisStep := STATE_STOP;
			END_IF
			(* check if error occured *)
			IF MC_MoveAbsolute_0.Error OR MC_ReadStatus_0.Errorstop THEN
				BasicControl.Status.ErrorID := MC_MoveAbsolute_0.ErrorID;
				MC_MoveAbsolute_0.Execute := TRUE;
				AxisStep := STATE_ERROR;
			END_IF

		(******************** START ADDITIVE MOVEMENT **********************)
		STATE_MOVE_ADDITIVE:  (* STATE: Start additive movement *)
			(* check if commanded distance is reached *)
			IF cmd <> CONST.AXIS.SETPOS AND cmd <> CONST.AXIS.STOP THEN
				MC_MoveAdditive_0.Execute := FALSE;
				cmdtmp := cmd;
				AxisStep := STATE_HALT;
				AxisStep := STATE_HALT;
			ELSIF MC_MoveAdditive_0.Done THEN
				MC_MoveAdditive_0.Execute := FALSE;
				cmdtmp := cmd;
				AxisStep := STATE_QUIT;
			ELSIF cmd = CONST.AXIS.STOP THEN
				MC_MoveAdditive_0.Execute := FALSE;
				MC_Stop_0( Execute := TRUE, Deceleration := verzoegerung);
				AxisStep := STATE_STOP;
			END_IF
			(* check if error occured *)
			IF MC_MoveAdditive_0.Error OR  MC_ReadStatus_0.Errorstop THEN
				BasicControl.Status.ErrorID := MC_MoveAdditive_0.ErrorID;
				MC_MoveAdditive_0.Execute := FALSE;
				AxisStep := STATE_ERROR;
			END_IF

		(******************** START VELOCITY MOVEMENT **********************)
		STATE_MOVE_VELOCITY:  (* STATE: Start velocity movement *)
			IF cmd <>  CONST.AXIS.MOVE_VELOCITY AND  cmd <> CONST.AXIS.STOP THEN
				MC_MoveVelocity_0.Execute := FALSE;
				cmdtmp := cmd;
				AxisStep := STATE_HALT;
			ELSIF MC_MoveVelocity_0.InVelocity THEN
				MC_MoveVelocity_0.Execute := FALSE;
				cmdtmp := cmd;
				AxisStep := STATE_QUIT;
			ELSIF cmd = CONST.AXIS.STOP THEN
				MC_MoveVelocity_0.Execute := FALSE;
				MC_Stop_0( Execute := TRUE, Deceleration := verzoegerung);
				AxisStep := STATE_STOP;
			END_IF
			(* check if error occured *)
			IF MC_MoveVelocity_0.Error OR MC_ReadStatus_0.Errorstop  THEN
				BasicControl.Status.ErrorID := MC_MoveVelocity_0.ErrorID;
				MC_MoveVelocity_0.Execute := FALSE;
				AxisStep := STATE_ERROR;
			END_IF

		(******************** FB-ERROR OCCURED *************************)
		STATE_ERROR:  (* STATE: Error *)
			(* check if FB indicates an axis error *)
			IF (MC_ReadAxisError_0.AxisErrorCount<>0) THEN
				AxisStep := STATE_ERROR_AXIS;
			ELSE
				IF (BasicControl.Command.ErrorAcknowledge = TRUE) THEN
					BasicControl.Command.ErrorAcknowledge := FALSE;
					BasicControl.Status.ErrorID := 0;
					(* reset axis if it is in axis state ErrorStop *)
					IF MC_ReadStatus_0.Errorstop AND MC_ReadStatus_0.Valid  THEN
						AxisStep := STATE_ERROR_RESET;
					ELSE
						(*AxisStep := STATE_WAIT;*)
						cmdtmp := cmd;
						AxisStep := STATE_QUIT;
					END_IF
				END_IF
			END_IF

		(******************** AXIS-ERROR OCCURED *************************)
		STATE_ERROR_AXIS:  (* STATE: Axis Error *)
			IF (MC_ReadAxisError_0.Valid) THEN
				err.set := TRUE;
				err.text := MC_ReadAxisError_0.DataObjectName;
				err.id :=  UINT_TO_DINT  (MC_ReadAxisError_0.AxisErrorID) ;
				IF (MC_ReadAxisError_0.AxisErrorID <> 0) THEN
					BasicControl.Status.ErrorID := MC_ReadAxisError_0.AxisErrorID;
				END_IF
				MC_ReadAxisError_0.Acknowledge := FALSE;
			(*	IF (BasicControl.Command.ErrorAcknowledge) THEN
					BasicControl.Command.ErrorAcknowledge := FALSE;
					(* acknowledge axis error *)
				IF cmd = CONST.AXIS.RESET THEN
					IF (MC_ReadAxisError_0.AxisErrorID <> 0) THEN
						MC_ReadAxisError_0.Acknowledge := TRUE;
						AxisStep := STATE_ERROR_RESET;
					END_IF
				END_IF
				IF (MC_ReadAxisError_0.AxisErrorCount = 0) THEN
					(* reset axis if it is in axis state ErrorStop *)
					BasicControl.Status.ErrorID := 0;
					IF ((MC_ReadStatus_0.Errorstop ) AND (MC_ReadStatus_0.Valid)) THEN
						AxisStep := STATE_ERROR_RESET;
					ELSE
						(*AxisStep := STATE_WAIT;*)
						cmdtmp := cmd;
						AxisStep := STATE_QUIT;
					END_IF
				ELSIF NOT MC_ReadAxisError_0.Error THEN
					cmdtmp := cmd;
					AxisStep := STATE_QUIT;
				END_IF
			ELSE
				AxisStep := STATE_WAIT; (* kein Fehler liegt vor*)
			END_IF

		(******************** RESET DONE *************************)
		STATE_ERROR_RESET:  (* STATE: Wait for reset done *)
			MC_Reset_0.Execute := TRUE;
			(* reset MC_Power.Enable if this FB is in Error*)
			IF (MC_Power_0.Error) THEN
				MC_Power_0.Enable := FALSE;
			END_IF
			IF(MC_Reset_0.Done)THEN
				MC_Reset_0.Execute := FALSE;
				cmdtmp := cmd;
				AxisStep := STATE_QUIT;
			ELSIF(MC_Reset_0.Error) THEN
				MC_Reset_0.Execute := FALSE;
				AxisStep := STATE_ERROR;
			END_IF
		(******************** SEQUENCE END *************************)
		STATE_QUIT:
			busy := FALSE;
			IF cmd = cmdtmp THEN
				busy := FALSE;
				cmd := CONST.AXIS.NOACTION;
				AxisStep := STATE_READY;
			ELSIF cmd <> CONST.AXIS.NOACTION THEN
				busy := FALSE;
				AxisStep := STATE_READY;
			END_IF

	END_CASE

(***************************************************************
        FUNCTION Block Calls
***************************************************************)

(************************** MC_POWER ****************************)
	MC_Power_0.Axis := AxisREF;  (* pointer to axis *)
	MC_Power_0();

	(************************** MC_HOME *****************************)
	MC_Home_0.Axis := AxisREF;
	MC_Home_0();

	(********************** MC_MOVEABSOLUTE *************************)
	MC_MoveAbsolute_0.Acceleration := BasicControl.Parameter.Acceleration;
	MC_MoveAbsolute_0.Deceleration := BasicControl.Parameter.Deceleration;
	MC_MoveAbsolute_0.Axis := AxisREF;
	MC_MoveAbsolute_0();

	(********************** MC_MOVEADDITIVE *************************)
	MC_MoveAdditive_0.Acceleration := BasicControl.Parameter.Acceleration;
	MC_MoveAdditive_0.Deceleration := BasicControl.Parameter.Deceleration;
	MC_MoveAdditive_0.Axis := AxisREF;
	MC_MoveAdditive_0();

	(********************** MC_MOVEVELOCITY *************************)
	MC_MoveVelocity_0.Acceleration  := BasicControl.Parameter.Acceleration;
	MC_MoveVelocity_0.Deceleration  := BasicControl.Parameter.Deceleration;
	MC_MoveVelocity_0.Axis := AxisREF;
	MC_MoveVelocity_0();

	(************************** MC_STOP *****************************)
	MC_Stop_0.Axis := AxisREF;
	MC_Stop_0();

	(***************************MC_HALT******************************)
	MC_Halt_0.Axis := AxisREF;
	MC_Halt_0();

	(************************** MC_RESET ****************************)
	MC_Reset_0.Axis := AxisREF;
	MC_Reset_0();

END_FUNCTION_BLOCK
```

#### Package Logical/Bibliothek/Counters - Paket

#### FB_Counter.st
```iecst
(********************************************************************
 * COPYRIGHT -- Microsoft
 ********************************************************************
 * Library: Bibliothek
 * Datei: FB_Counter.st
 * Autor: okrebs
 * Erstellt: 31. Juli 2014
 ********************************************************************
 * Implementierung der Library Bibliothek
 ********************************************************************)

(* TODO: Bitte Kommentar hier einfügen *)
FUNCTION_BLOCK FB_Counter

	R_trig(CLK := triggerInput);
//
//	IF counter = 0 THEN
//		counter := setPieces;
//	ELSE
	IF (*counter = setPieces*)FALSE THEN // OKrebs 27.04.17
		counter := 0;
	ELSE
		IF R_trig.Q OR countPlusVisu THEN
			(*counter := counter - 1;*)
			counter := counter + 1;
		ELSIF countMinusVisu THEN
			counter := counter - 1;
//			IF counter = 0 THEN
//				counterTemp := counterTemp + 1;
//			END_IF
		END_IF
	END_IF

	IF reset THEN
		counterTemp := counter;
		counter := 0;
	END_IF

END_FUNCTION_BLOCK
```

#### FB_Counters.st
```iecst
(********************************************************************
 * COPYRIGHT -- Microsoft
 ********************************************************************
 * Library: Bibliothek
 * Datei: FB_Counters.st
 * Autor: okrebs
 * Erstellt: 31. Juli 2014
 ********************************************************************
 * Implementierung der Library Bibliothek
 ********************************************************************)

(* TODO: Bitte Kommentar hier einfügen *)
FUNCTION_BLOCK FB_Counters
//	IF counter1.counter >= counter1.setPieces OR  counter2.counter >= counter2.setPieces OR counter3.counter >= counter3.setPieces
//	 OR counter4.counter >= counter4.setPieces OR 	counter5.counter >= counter5.setPieces OR counter6.counter >= counter6.setPieces
//	 OR counter7.counter >= counter7.setPieces OR 	counter8.counter >= counter8.setPieces OR counter9.counter >= counter9.setPieces AND NOT reset THEN
//		reset := TRUE;
//	END_IF

//	IF  setPieces <= counter2.counter OR setPieces <= counter4.counter OR setPieces <= counter6.counter OR
//		setPieces <= counter8.counter THEN
//		Nitto_Table_Full := TRUE;
//	END_IF
// new //26.07.18 // OKrebs
	IF  setPieces <= counter2.counter AND setPieces <= counter4.counter AND setPieces <= counter6.counter AND
		setPieces <= counter8.counter THEN
		Nitto_Table_Full := TRUE;
	END_IF

// new // OKrebs // 27.04.17
//	IF  setPieces <= counter2.counter AND setPieces <= counter4.counter AND setPieces <= counter6.counter AND
//		setPieces <= counter8.counter THEN
//		Nitto_Table_Full := TRUE;
//	END_IF
// end new

	IF EDGEPOS((5 <= counter2.counter AND 10 >= counter2.counter) OR
		(5 <= counter4.counter AND 10 >= counter4.counter) OR
		(5 <= counter6.counter AND 10 >= counter6.counter) OR
		(5 <= counter8.counter AND 10 >= counter8.counter) OR
		manualButton OR visureset)	THEN
		Nitto_Table_Full := FALSE;
	END_IF

//	IF visureset OR reset OR EDGEPOS(Nitto_Table_Full) OR manualButton THEN
//		reset := TRUE;
//		visureset := FALSE;
//	ELSIF NOT visureset OR NOT manualButton OR EDGENEG(Nitto_Table_Full)THEN
//		reset := FALSE;
//	END_IF

	TON_reset.PT := T#500ms;

	IF EDGEPOS(visureset OR Nitto_Table_Full OR manualButton) THEN
		TON_reset.IN := TRUE;
	END_IF

	reset := TON_reset.Q;

	counter1(reset := reset, setPieces := setPieces);
	counter2(reset := reset, setPieces := setPieces);
	counter3(reset := reset, setPieces := setPieces);
	counter4(reset := reset, setPieces := setPieces);
	counter5(reset := reset, setPieces := setPieces);
	counter6(reset := reset, setPieces := setPieces);
	counter7(reset := reset, setPieces := setPieces);
	counter8(reset := reset, setPieces := setPieces);
	counter9(reset := reset, setPieces := setPieces);
	IF validpieces <= counter1.counter OR validpieces <= counter2.counter
		OR validpieces <= counter3.counter OR validpieces <= counter4.counter OR
		validpieces <= counter4.counter OR validpieces <= counter5.counter OR validpieces <= counter6.counter OR
		validpieces <= counter7.counter OR validpieces <= counter8.counter OR validpieces <= counter9.counter THEN
		valid := TRUE;
	//	Nitto_Table_Full := TRUE;
		(* für ein akusteisches Signal*)
	ELSE
		valid := FALSE;
	END_IF

	IF TON_reset.Q THEN
		TON_reset.IN := FALSE;
	END_IF

	TON_reset();

	// 26.07.18 // OKrebs // Programm fuer die neue Ampel
	TON_Nitto_Table_Full(IN := Nitto_Table_Full, PT := T#1s);
	TP_GreenLampOut.PT := T#4s;

	IF EDGEPOS(TON_Nitto_Table_Full.Q) THEN
		IF setPieces <> counter2.counterTemp OR setPieces <> counter4.counterTemp OR setPieces <> counter6.counterTemp OR
		setPieces <> counter8.counterTemp THEN
		RedLampOut := TRUE;
		ELSE
		TP_GreenLampOut.IN := TRUE;
		END_IF
	END_IF

	IF VisuOKButton THEN
		RedLampOut := FALSE;
		GreenLampOut := FALSE;
	END_IF

	GreenLampOut := TP_GreenLampOut.Q;

	IF EDGENEG(TP_GreenLampOut.Q) THEN
		TP_GreenLampOut.IN := FALSE;
	END_IF

	TP_GreenLampOut();

END_FUNCTION_BLOCK
```

#### FB_SprayCtrl.st
```iecst
(********************************************************************
 * COPYRIGHT -- Nitto
 ********************************************************************
 * Library: Bibliothek
 * Datei: FB_SprayCtrl.st
 * Autor: s_spilker
 * Erstellt: 11. September 2014
 ********************************************************************
 * Implementierung der Library Bibliothek
 ********************************************************************)

(* TODO: Bitte Kommentar hier einfügen *)
FUNCTION_BLOCK FB_SprayCtrl
	machineaxis();

	IF machineaxis.MC_ReadActualVelocity_0.Velocity > 100 THEN // 25.07.18 //OKrebs damit Sprueanlage nicht im Stand spruet

	time1.PT :=	REAL_TO_TIME (length1*1000 (*length1*1000*1000 / machineaxis.MC_ReadActualVelocity_0.Velocity*));
	time2.PT := REAL_TO_TIME (length2*1000*1000 / machineaxis.MC_ReadActualVelocity_0.Velocity);
	END_IF

//	R_TRIG_0(CLK := machineaxis.MC_ReadStatus_0.ContinuousMotion);
//	IF R_TRIG_0.Q THEN
//		time1.IN := FALSE;
//		time2.IN := FALSE;
//	END_IF;

//	time1.PT := T#1s;
//	time2.PT := T#2s;
	time1();
	time2();
	F_TRIG_1(CLK := time1.Q);
	F_TRIG_2(CLK := time2.Q);
	//	time_tof := REAL_TO_TIME(spraytime);
//	timer_tof(PT := time_tof);
//	test :=  fmod(machineaxis.MC_ReadActualPosition_0.Position,lenght);
	//	test1 := modf(machineaxis.MC_ReadActualPosition_0.Position,lenght);
	(*test1 := machineaxis.MC_ReadActualPosition_0.Position;*)
//	rtrig();
	IF length1 = 0 THEN
		valveout := FALSE;
	ELSE
		IF machineaxis.MC_ReadStatus_0.ContinuousMotion THEN

			CASE pulse OF

				1: (*AN*)
				time1.IN := TRUE;
				valveout := TRUE;
					IF F_TRIG_1.Q THEN
					time1.IN := FALSE;
					pulse := 2;
					END_IF

				2: (*AUS*)
				time2.IN := TRUE;
				valveout := FALSE;
					IF F_TRIG_2.Q THEN
					time2.IN := FALSE;
					pulse := 1;
					END_IF

			END_CASE

//			IF lenght - 80 < fmod(machineaxis.MC_ReadActualPosition_0.Position,lenght ) THEN
//				rtrig.CLK := TRUE;
//			END_IF
//
//
//			IF rtrig.Q THEN
//				timer_tof.IN := TRUE;
//				test1 := test1 + 1;
//				(*rtrig.CLK := FALSE;*)
//			END_IF
//			IF timer_tof.Q THEN
//				rtrig.CLK := FALSE;
//				timer_tof.IN := FALSE;
//			END_IF
//			valveout :=	timer_tof.Q;
		ELSE
			valveout := FALSE;
			time1.IN := FALSE;
			time2.IN := FALSE;
		END_IF
	END_IF
END_FUNCTION_BLOCK
```

#### FB_AxisCtrl_new.st
```iecst
(********************************************************************
 * COPYRIGHT -- Nitto
 ********************************************************************
 * Library: Bibliothek
 * Datei: FB_AxisCtrl_new.st
 * Autor: s_spilker
 * Erstellt: 9. November 2015
 ********************************************************************
 * Implementierung der Library Bibliothek
 ********************************************************************)

(* TODO: Bitte Kommentar hier einfügen *)
FUNCTION_BLOCK FB_AxisCtrl_new

(***************************************************************
        Control Sequence
***************************************************************)
(* status information is read before the step sequencer to attain a shorter reaction time *)
(************************ MC_READSTATUS *************************)
	MC_ReadStatus_0.Enable :=  NOT MC_ReadStatus_0.Error;
	MC_ReadStatus_0.Axis := AxisREF;
	MC_ReadStatus_0();
	(********************MC_BR_READDRIVESTATUS***********************)
	MC_BR_ReadDriveStatus_0.Enable := NOT(MC_BR_ReadDriveStatus_0.Error);
	MC_BR_ReadDriveStatus_0.Axis := AxisREF;
	MC_BR_ReadDriveStatus_0.AdrDriveStatus := ADR(BasicControl.Status.DriveStatus);
	MC_BR_ReadDriveStatus_0();
	(******************** MC_READACTUALPOSITION *********************)
	MC_ReadActualPosition_0.Enable := (NOT(MC_ReadActualPosition_0.Error));
	MC_ReadActualPosition_0.Axis := AxisREF;
	MC_ReadActualPosition_0();//B&R kennt wohl Ausgagstypen nicht

	(******************** MC_READACTUALVELOCITY *********************)
	MC_ReadActualVelocity_0.Enable := (NOT(MC_ReadActualVelocity_0.Error));
	MC_ReadActualVelocity_0.Axis := AxisREF;
	MC_ReadActualVelocity_0();

	(*********************+*Parameter schreiben**********************)
	(************************ MC_READAXISERROR **********************)
	MC_ReadAxisError_0.Enable := NOT(MC_ReadAxisError_0.Error);
	MC_ReadAxisError_0.Axis := AxisREF;
	MC_ReadAxisError_0.DataAddress := ADR(BasicControl.Status.ErrorText);
	MC_ReadAxisError_0.DataLength := SIZEOF(BasicControl.Status.ErrorText);
	MC_ReadAxisError_0.DataObjectName := 'acp10etxde';
	MC_ReadAxisError_0();
	(* central monitoring OF stop command attains a shorter reaction TIME in CASE OF emergency stop *)
	(******************CHECK FOR STOP COMMAND************************)
	CASE AxisStep OF

//		******************* WAIT ************************
		STATE_WAIT:  (* STATE: Wait *)
			AxisStep := STATE_QUIT;

//		(********************Virtuelle Achse einschalten****)
		STATE_VAXIS_ON:

			IF MC_BR_ReadDriveStatus_0.Valid THEN
				cmdtmp := Cmd;
				AxisStep := STATE_QUIT;
			END_IF
		(******************** POWER ON **********************)
		STATE_POWER_ON:  (* STATE: Power on *)
			(*MC_Power_0.Enable := TRUE;*)
			MC_Power_0.Axis := AxisREF;
			MC_Power_0();
			IF BasicControl.Status.DriveStatus.ControllerReady AND	Cmd = CONST.AXIS.POWER_ON
				AND NOT MC_Power_0.Status AND NOT MC_Power_0.Error THEN
				MC_Power_0.Enable := TRUE; (*erster Anlauf*)
					cmdtmp := Cmd;
			ELSIF MC_Power_0.Error AND cmdtmp = Cmd THEN
					MC_Power_0.Enable := FALSE ;(* if a power error occured go to error state *)
					Cmd := CONST.AXIS.RESET;
					err.set := TRUE;
					err.fnc := 'FB_AxisCtrl';
					err.id  := MC_Power_0.ErrorID;
					err.state := AxisStep;
					AxisStep := STATE_ERROR_RESET;
			ELSIF 	MC_Power_0.Status AND NOT MC_Power_0.Error THEN
					cmdtmp := Cmd;
					AxisStep := STATE_QUIT;
			ELSIF MC_ReadStatus_0.Errorstop THEN (*24.07.14*)
					BasicControl.Status.ErrorID := MC_Power_0.ErrorID;
					err.set := TRUE;
					err.fnc := 'FB_AxisCtrl';
					err.id  := MC_Power_0.ErrorID;;
					err.state := AxisStep;
					AxisStep := STATE_ERROR;
			END_IF
		(******************* POWER OFF *********************)
		STATE_POWER_OFF:  (* STATE: Power off *)
			MC_Power_0.Axis := AxisREF;
			MC_Power_0.Enable := FALSE;
			MC_Power_0();
			IF NOT MC_Power_0.Status AND NOT MC_Power_0.Busy  THEN
				cmdtmp := Cmd;
				AxisStep := STATE_QUIT;
			END_IF
			(* if a power error occured go to error state *)
			IF MC_Power_0.Error  THEN
				BasicControl.Status.ErrorID := MC_Power_0.ErrorID;
				err.set := TRUE;
				err.fnc := 'FB_AxisCtrl';
				err.id  := MC_Power_0.ErrorID;
				err.state := AxisStep;
				AxisStep := STATE_ERROR;
			END_IF
		(******************** READY **********************)
		STATE_READY:  (* STATE: Waiting for commands *)
			IF Cmd <> CONST.AXIS.NOACTION THEN
					busy := TRUE;
					(*cmdtmp:= Cmd; *)
					IF Cmd = CONST.AXIS.RESET THEN
						AxisStep := STATE_ERROR_RESET;
					ELSIF Cmd = CONST.AXIS.STOP  THEN
						MC_Stop_0.Execute := TRUE;
						MC_Stop_0.Deceleration := Deceleration;
						AxisStep := STATE_STOP;
					ELSIF Cmd = CONST.AXIS.JOG_NEG THEN
						MC_BR_JogVelocity_0.Enable := TRUE;
						MC_BR_JogVelocity_0.Velocity := 16666*Velocity;
						MC_BR_JogVelocity_0.Acceleration := Acceleration;
						MC_BR_JogVelocity_0.Deceleration  := Deceleration;
						MC_BR_JogVelocity_0.JogPositive := FALSE;
						MC_BR_JogVelocity_0.JogNegative := TRUE;
						AxisStep := STATE_JOG_NEGATIVE;
					ELSIF Cmd = CONST.AXIS.JOG_POS THEN
						MC_BR_JogVelocity_0.Enable := TRUE;
						MC_BR_JogVelocity_0.Velocity := 16666*Velocity;
						MC_BR_JogVelocity_0.Acceleration := Acceleration;
						MC_BR_JogVelocity_0.Deceleration  := Deceleration;
						MC_BR_JogVelocity_0.JogPositive := TRUE;
						MC_BR_JogVelocity_0.JogNegative := FALSE;
						AxisStep := STATE_JOG_POSITIVE;
					ELSIF Cmd = CONST.AXIS.SETPOS THEN
						MC_MoveAbsolute_0(Execute := TRUE, Position := Position, Velocity := 16666*Velocity, Acceleration := Acceleration,
										Deceleration  := BasicControl.Parameter.Deceleration, Direction := mcPOSITIVE_DIR);
						AxisStep := STATE_MOVE_ABSOLUTE;
					ELSIF Cmd = CONST.AXIS.SETPOSREL THEN
						MC_BR_JogLimitPosition_0.Enable := TRUE;
						MC_BR_JogLimitPosition_0.Velocity := 16666*Velocity;
						MC_BR_JogLimitPosition_0.Acceleration := Acceleration;
						MC_BR_JogLimitPosition_0.Deceleration := Deceleration;
						MC_BR_JogLimitPosition_0.LastPosition := Position;
//						MC_BR_JogLimitPosition_0.FirstPosition := - 2147483647;//nicht vergessen
						MC_BR_JogLimitPosition_0.JogPositive  := TRUE;
						MC_BR_JogLimitPosition_0.JogNegative  := FALSE;
						AxisStep := STATE_MOVE_ADDITIVE;
					ELSIF Cmd = CONST.AXIS.MOVE_VELOCITY THEN
							MC_MoveVelocity_0(Execute := TRUE, Velocity := 16666*Velocity, Acceleration := Acceleration,
												Deceleration  := Deceleration,	Direction := mcPOSITIVE_DIR);
						AxisStep := STATE_MOVE_VELOCITY;
					ELSIF Cmd = CONST.AXIS.SETPOSREL_NOLIMIT THEN
						MC_MoveAdditive_0(Execute := TRUE, Distance := Position, Velocity := 16666*Velocity, Acceleration := Acceleration,
										Deceleration  := Deceleration);
						AxisStep := STATE_MOVE_ADDITIVELIMIT;
					ELSIF Cmd = CONST.AXIS.MOVE_CYCLIC_VELOCITY THEN
						MC_BR_JogVelocity_0.Enable := TRUE;
						MC_BR_JogVelocity_0.Velocity := 16666*Velocity;
						MC_BR_JogVelocity_0.Acceleration := Acceleration;
						MC_BR_JogVelocity_0.Deceleration  := Deceleration;
						MC_BR_JogVelocity_0.JogPositive := TRUE;
						MC_BR_JogVelocity_0.JogNegative := FALSE;
						AxisStep := STATE_MOVE_CYCLIC_VELOCITY;
					ELSIF  Cmd = CONST.AXIS.CALIBR THEN
						MC_Home_0.Execute := TRUE;
						MC_Home_0.Position := BasicControl.Parameter.HomePosition;
						MC_Home_0.HomingMode := BasicControl.Parameter.HomeMode;
						AxisStep := STATE_HOME;
					ELSIF   Cmd = CONST.AXIS.POWER_OFF THEN
						AxisStep := STATE_POWER_OFF;
					ELSIF   Cmd = CONST.AXIS.POWER_ON THEN
						AxisStep := STATE_POWER_ON;
					END_IF
			ELSE
				busy := FALSE;
			END_IF
		(******************** HOME **********************)
		STATE_HOME:  (* STATE: start homing process *)
//			MC_Home_0.Axis := AxisREF;
//			MC_Home_0();
			IF MC_Home_0.Done AND Cmd = CONST.AXIS.CALIBR THEN
				MC_Home_0.Execute := FALSE;
				BasicControl.AxisState.Homed := TRUE;
			ELSIF BasicControl.AxisState.Homed  AND NOT MC_Home_0.Done THEN // Referenzierung beendet
				cmdtmp := Cmd;
				AxisStep := STATE_QUIT;
			ELSIF Cmd <> CONST.AXIS.CALIBR THEN //da nur der MC_Stop den Zustand Homing unterbrechen kann
				MC_Home_0.Execute 		:= FALSE;
				MC_Stop_0.Deceleration 	:= Deceleration;
				MC_Stop_0.Execute 		:= TRUE;
				AxisStep := STATE_STOP;
			ELSIF MC_Home_0.CommandAborted AND Cmd = CONST.AXIS.CALIBR THEN
				MC_Home_0.Execute := FALSE;
				AxisStep := STATE_READY;
			END_IF
			(* if a homing error occured go to error state *)
			IF MC_Home_0.Error  THEN
				MC_Home_0.Execute := FALSE;
				BasicControl.Status.ErrorID := MC_Home_0.ErrorID;
				err.set := TRUE;
				err.fnc := 'MC_Home_0';
				err.id  := MC_Home_0.ErrorID;
				err.text := BasicControl.Status.ErrorText[0];
				err.state := AxisStep;
				AxisStep := STATE_ERROR;
			END_IF

		(***********************HALT_MOVEMENT***************************)
		STATE_HALT:   (* STATE: Halt movement *)
			MC_Halt_0.Deceleration := Deceleration;
			MC_Halt_0.Execute := TRUE;
			IF MC_Halt_0.Done THEN
				MC_Halt_0.Execute := FALSE;
				cmdtmp := Cmd;
				AxisStep := STATE_QUIT;
			END_IF
			(* check if error occured *)
			IF MC_Halt_0.Error  THEN
				BasicControl.Status.ErrorID := MC_Halt_0.ErrorID;
				MC_Halt_0.Execute := FALSE;
				err.set := TRUE;
				err.fnc := 'FB_AxisCtrl';
				err.id  := MC_Halt_0.ErrorID;
				err.state := AxisStep;
				AxisStep := STATE_ERROR;
			END_IF

		(*********************** STOP MOVEMENT *************************)
		STATE_STOP:  (* STATE: Stop movement *)
		(*	MC_Stop_0.Execute := TRUE;*)
			(* if axis is stopped go to ready state *)
			MC_BR_JogVelocity_0.Axis := AxisREF;
			MC_BR_JogVelocity_0.Velocity := 16666*Velocity;
			MC_BR_JogVelocity_0();
			MC_BR_JogLimitPosition_0.Axis := AxisREF;
			MC_BR_JogLimitPosition_0.Enable := FALSE;
			MC_BR_JogLimitPosition_0();
			IF MC_Stop_0.Done OR MC_ReadStatus_0.StandStill THEN
				MC_Stop_0.Execute := FALSE;
				cmdtmp := Cmd;
				AxisStep := STATE_QUIT;
//			ELSIF MC_ReadStatus_0.Disabled THEN
//				MC_Stop_0.Execute := FALSE;
//				cmdtmp := Cmd;
//				AxisStep := STATE_QUIT;
			END_IF
			(* check if error occured *)
			IF MC_Stop_0.Error THEN
				BasicControl.Status.ErrorID := MC_Stop_0.ErrorID;
				MC_Stop_0.Execute := FALSE;
				err.set := TRUE;
				err.fnc := 'FB_AxisCtrl';
				err.id  := MC_Stop_0.ErrorID;
				err.state := AxisStep;
				AxisStep := STATE_ERROR;
			ELSIF MC_ReadStatus_0.Errorstop THEN
		 		MC_Stop_0.Execute := FALSE;
				err.set := TRUE;
				err.fnc := 'FB_AxisCtrl';
				err.text  := BasicControl.Status.ErrorText[0];
				err.state := AxisStep;
				AxisStep := STATE_ERROR;
			END_IF

		(******************** START JOG MOVEMENT POSITVE **********************)
		STATE_JOG_POSITIVE:  (* STATE: Start jog movement in positive direction *)
			MC_BR_JogVelocity_0.Axis := AxisREF;
			MC_BR_JogVelocity_0.Velocity := 16666*Velocity;
			MC_BR_JogVelocity_0();

			IF Cmd <> CONST.AXIS.JOG_POS  AND Cmd <> CONST.AXIS.STOP THEN
				MC_BR_JogVelocity_0.Enable := FALSE;
				cmdtmp := Cmd;
				IF NOT MC_BR_JogVelocity_0.Busy THEN
					AxisStep := STATE_QUIT;
				END_IF
			ELSIF Cmd = CONST.AXIS.STOP THEN
				MC_BR_JogVelocity_0.Enable := FALSE;
				MC_Stop_0( Execute := TRUE, Deceleration := Deceleration);
				AxisStep := STATE_STOP;
			END_IF
			IF MC_BR_JogVelocity_0.Error THEN
				BasicControl.Status.ErrorID := MC_BR_JogVelocity_0.ErrorID;
				MC_BR_JogVelocity_0.Enable := FALSE;
				err.set := TRUE;
				err.fnc := 'FB_AxisCtrl';
				err.id := MC_BR_JogVelocity_0.ErrorID;
				err.state := AxisStep;
				AxisStep := STATE_ERROR;
			END_IF

		(******************** START JOG MOVEMENT NEGATIVE **********************)
		STATE_JOG_NEGATIVE:  (* STATE: Start jog movement in negative direction *)
			MC_BR_JogVelocity_0.Axis := AxisREF;
			MC_BR_JogVelocity_0.Velocity := 16666*Velocity;
			MC_BR_JogVelocity_0();
			IF Cmd <> CONST.AXIS.JOG_NEG AND Cmd <> CONST.AXIS.STOP  THEN
				MC_BR_JogVelocity_0.Enable := FALSE;
				cmdtmp := Cmd;
				IF NOT MC_BR_JogVelocity_0.Busy THEN
					AxisStep := STATE_QUIT;
				END_IF
			ELSIF Cmd = CONST.AXIS.STOP THEN
				MC_BR_JogVelocity_0.Enable := FALSE;
				MC_Stop_0( Execute := TRUE, Deceleration := Deceleration);
				AxisStep := STATE_STOP;
			END_IF
			IF MC_BR_JogVelocity_0.Error THEN
				BasicControl.Status.ErrorID := MC_BR_JogVelocity_0.ErrorID;
				MC_BR_JogVelocity_0.Enable := FALSE;
				err.set := TRUE;
				err.fnc := 'FB_AxisCtrl';
				err.id := MC_BR_JogVelocity_0.ErrorID;
				err.state := AxisStep;
				AxisStep := STATE_ERROR;
			END_IF

		(******************** START ABSOLUTE MOVEMENT **********************)
		STATE_MOVE_ABSOLUTE:  (* STATE: Start absolute movement *)
			(* check if commanded position is reached *)
			IF Cmd <> CONST.AXIS.SETPOS AND Cmd <> CONST.AXIS.STOP THEN
				MC_MoveAbsolute_0.Execute := FALSE;
				cmdtmp := Cmd;
				AxisStep := STATE_HALT;
			ELSIF MC_MoveAbsolute_0.Done  THEN
				MC_MoveAbsolute_0.Execute := FALSE;
				cmdtmp := Cmd;
				AxisStep := STATE_QUIT;
			ELSIF Cmd = CONST.AXIS.STOP THEN
				MC_MoveAbsolute_0.Execute := FALSE;
				MC_Stop_0( Execute := TRUE, Deceleration := Deceleration);
				AxisStep := STATE_STOP;
			END_IF
			(* check if error occured *)
			IF MC_MoveAbsolute_0.Error THEN
				BasicControl.Status.ErrorID := MC_MoveAbsolute_0.ErrorID;
				MC_MoveAbsolute_0.Execute := TRUE;
				err.set := TRUE;
				err.fnc := 'FB_AxisCtrl';
				err.id  := MC_MoveAbsolute_0.ErrorID;
				err.state := AxisStep;
				AxisStep := STATE_ERROR;
			END_IF

		(******************** START ADDITIVE MOVEMENT **********************)
		STATE_MOVE_ADDITIVE:  (* STATE: Start additive movement *)
			(* check if commanded distance is reached *)
			//mit MC_MoveAdditive kann man die Geschwindigkeit nicht permanent ändern
			MC_BR_JogLimitPosition_0.Axis := AxisREF;
			MC_BR_JogLimitPosition_0.Velocity := 16666*Velocity;
			MC_BR_JogLimitPosition_0();
			IF MC_BR_JogLimitPosition_0.LimitReached THEN
				MC_BR_JogLimitPosition_0.Enable := FALSE;
				cmdtmp := Cmd;
			ELSIF NOT MC_BR_JogLimitPosition_0.Busy  THEN
					AxisStep := STATE_QUIT;
			ELSIF Cmd = CONST.AXIS.STOP THEN
				MC_BR_JogLimitPosition_0.Enable := FALSE;
				MC_Stop_0( Execute := TRUE, Deceleration := Deceleration);
				AxisStep := STATE_STOP;
			END_IF
			IF MC_BR_JogLimitPosition_0.Error THEN
				BasicControl.Status.ErrorID := MC_BR_JogLimitPosition_0.ErrorID;
				MC_BR_JogLimitPosition_0.Enable := FALSE;
				err.set := TRUE;
				err.fnc := 'FB_AxisCtrl';
				err.id := MC_BR_JogLimitPosition_0.ErrorID;
				err.text := BasicControl.Status.ErrorText[0];
				err.state := AxisStep;
				AxisStep := STATE_ERROR;
			END_IF

		STATE_MOVE_ADDITIVELIMIT:
			IF Cmd<> CONST.AXIS.SETPOSREL_NOLIMIT  THEN
				MC_MoveAdditive_0.Execute := FALSE;
				cmdtmp := Cmd;
				AxisStep := STATE_HALT;
			ELSIF MC_MoveAdditive_0.Done  THEN
				MC_MoveAdditive_0.Execute := FALSE;
					(*AxisStep := STATE_READY;*)
					cmdtmp := Cmd;
					AxisStep := STATE_QUIT;
			END_IF
			(* check if error occured *)
			IF (MC_MoveAdditive_0.Error = TRUE) THEN
				BasicControl.Status.ErrorID := MC_MoveAdditive_0.ErrorID;
				MC_MoveAdditive_0.Execute := FALSE;
				AxisStep := STATE_ERROR;
			END_IF
			CyclicVelocity  := 16666*Velocity;
			MC_BR_CyclicWrite_0.Axis		:= AxisREF;
			MC_BR_CyclicWrite_0.DataAddress	:= ADR(CyclicVelocity);
			MC_BR_CyclicWrite_0.DataType	:= ncPAR_TYP_REAL;
			MC_BR_CyclicWrite_0.ParID		:= ACP10PAR_VAR_R4_0 + 0;
			MC_BR_CyclicWrite_0();

		(******************** START VELOCITY MOVEMENT **********************)
		STATE_MOVE_VELOCITY:  (* STATE: Start velocity movement *)
			IF Cmd <>  CONST.AXIS.MOVE_VELOCITY  AND Cmd <> CONST.AXIS.STOP THEN
				MC_MoveVelocity_0.Execute := FALSE;
				cmdtmp := Cmd;
				AxisStep := STATE_HALT;
			ELSIF MC_MoveVelocity_0.InVelocity THEN
				MC_MoveVelocity_0.Execute := FALSE;
				cmdtmp := Cmd;
				AxisStep := STATE_QUIT;
			ELSIF Cmd = CONST.AXIS.STOP THEN
				MC_MoveVelocity_0.Execute := FALSE;
				MC_Stop_0( Execute := TRUE, Deceleration := Deceleration);
				AxisStep := STATE_STOP;
			END_IF
			(* check if error occured *)
			IF MC_MoveVelocity_0.Error THEN
				BasicControl.Status.ErrorID := MC_MoveVelocity_0.ErrorID;
				MC_MoveVelocity_0.Execute := FALSE;
				err.set := TRUE;
				err.fnc := 'FB_AxisCtrl';
				err.id  := MC_MoveVelocity_0.ErrorID;
				err.state := AxisStep;
				AxisStep := STATE_ERROR;
			END_IF

		STATE_MOVE_CYCLIC_VELOCITY:
			MC_BR_JogVelocity_0.Axis := AxisREF;
			MC_BR_JogVelocity_0.Velocity := 16666*Velocity;
			MC_BR_JogVelocity_0();
			IF Cmd <> CONST.AXIS.MOVE_CYCLIC_VELOCITY AND Cmd <> CONST.AXIS.STOP THEN
				MC_BR_JogVelocity_0.Enable := FALSE;
				cmdtmp := Cmd;
				IF NOT MC_BR_JogVelocity_0.Busy THEN
					AxisStep := STATE_QUIT;
				END_IF
			ELSIF Cmd = CONST.AXIS.STOP THEN
				MC_BR_JogVelocity_0.Enable := FALSE;
				MC_Stop_0( Execute := TRUE, Deceleration := Deceleration);
				AxisStep := STATE_STOP;
			END_IF
			IF MC_BR_JogVelocity_0.Error THEN
				BasicControl.Status.ErrorID := MC_BR_JogVelocity_0.ErrorID;
				MC_BR_JogVelocity_0.Enable := FALSE;
				err.set := TRUE;
				err.fnc := 'FB_AxisCtrl';
				err.id := MC_BR_JogVelocity_0.ErrorID;
				err.state := AxisStep;
				AxisStep := STATE_ERROR;
			END_IF

		(******************** FB-ERROR OCCURED *************************)

		STATE_ERROR:  (* STATE: Error *)
			(* check if FB indicates an axis error *)
			err();
			IF MC_ReadAxisError_0.AxisErrorCount<>0 THEN
				AxisStep := STATE_ERROR_AXIS;
			ELSE
				IF MC_ReadStatus_0.Errorstop AND MC_ReadStatus_0.Valid  THEN
					AxisStep := STATE_ERROR_AXIS;
				ELSIF Cmd = CONST.AXIS.RESET THEN
					cmdtmp := Cmd;
					AxisStep := STATE_ERROR_RESET;
				END_IF
			END_IF

		(******************** AXIS-ERROR OCCURED *************************)
		STATE_ERROR_AXIS:  (* STATE: Axis Error *)
			IF MC_ReadAxisError_0.Valid THEN
				err.set := TRUE;
				err.text := BasicControl.Status.ErrorText[0];
				err.id :=  UINT_TO_DINT  (MC_ReadAxisError_0.AxisErrorID) ;
				err();
				IF MC_ReadAxisError_0.AxisErrorID <> 0 THEN
						BasicControl.Status.ErrorID := MC_ReadAxisError_0.AxisErrorID;
				END_IF
				MC_ReadAxisError_0.Acknowledge := FALSE;
				IF Cmd = CONST.AXIS.RESET THEN
					IF MC_ReadAxisError_0.AxisErrorID <> 0 THEN
						MC_ReadAxisError_0.Acknowledge := TRUE;
						AxisStep := STATE_ERROR_RESET;
					END_IF
				END_IF
				IF MC_ReadAxisError_0.AxisErrorCount = 0 THEN
					(* reset axis if it is in axis state ErrorStop *)
					BasicControl.Status.ErrorID := 0;
					IF MC_ReadStatus_0.Errorstop AND MC_ReadStatus_0.Valid THEN
						AxisStep := STATE_ERROR_RESET;
					ELSE
						cmdtmp := Cmd;
						AxisStep := STATE_QUIT;
					END_IF
				ELSIF NOT MC_ReadAxisError_0.Error THEN
						cmdtmp := Cmd;
						AxisStep := STATE_QUIT;
				END_IF
			ELSE
				AxisStep := STATE_WAIT; (* kein Fehler liegt vor*)
			END_IF

		(******************** RESET DONE *************************)
		STATE_ERROR_RESET:  (* STATE: Wait for reset done *)
			MC_Reset_0.Execute := TRUE;
			MC_Power_0.Axis := AxisREF;
			MC_Power_0();
			MC_Home_0.Axis := AxisREF;
			MC_Home_0.Execute := FALSE;
			MC_Home_0();
			err.reset := TRUE;
			err();
			(* reset MC_Power.Enable if this FB is in Error*)
			IF MC_Power_0.Error THEN
				MC_Power_0.Enable := FALSE;
			END_IF
			IF MC_Reset_0.Done THEN
				MC_Reset_0.Execute := FALSE;
				cmdtmp := Cmd;
				AxisStep := STATE_QUIT;
			ELSIF MC_Reset_0.Error THEN
				MC_Reset_0.Execute := FALSE;
				AxisStep := STATE_ERROR;
			END_IF

		(******************** SEQUENCE END *************************)
		STATE_QUIT:
//
//			busy := FALSE;
//			IF Cmd = cmdtmp THEN
//				busy := FALSE;
//				Cmd := CONST.AXIS.NOACTION;
//				AxisStep := STATE_READY;
//			ELSIF Cmd <> CONST.AXIS.NOACTION THEN
//				AxisStep := STATE_READY;
//			END_IF
		busy:=FALSE;
		IF Cmd <> cmdtmp THEN
			IF Cmd = CONST.AXIS.RESET THEN
				busy := TRUE;
				AxisStep := STATE_ERROR_RESET;
			ELSIF Cmd = CONST.AXIS.STOP THEN
				MC_Stop_0( Execute := TRUE, Deceleration := Deceleration);
				busy := TRUE;
				AxisStep := STATE_STOP;
			ELSE
				busy := FALSE;
				AxisStep := STATE_READY;
			END_IF
		ELSE
			Cmd := CONST.AXIS.NOACTION;
			AxisStep := STATE_READY;
		END_IF
	END_CASE

(***************************************************************
        FUNCTION Block Calls
***************************************************************)

(************************** MC_POWER ****************************)
//	MC_Power_0.Axis := AxisREF;  (* pointer to axis *)
//	MC_Power_0();
	(************************** MC_HOME *****************************)
	MC_Home_0.Axis := AxisREF;
	MC_Home_0();
	(********************** MC_MOVEABSOLUTE *************************)
	MC_MoveAbsolute_0.Acceleration := Acceleration;
	MC_MoveAbsolute_0.Deceleration := Deceleration;
	MC_MoveAbsolute_0.Axis := AxisREF;
	MC_MoveAbsolute_0();
	(********************** MC_MOVEADDITIVE *************************)
	MC_MoveAdditive_0.Acceleration := Acceleration;
	MC_MoveAdditive_0.Deceleration := Deceleration;
	MC_MoveAdditive_0.Axis := AxisREF;
	MC_MoveAdditive_0();
	(********************** MC_MOVEVELOCITY *************************)
	MC_MoveVelocity_0.Acceleration  := Acceleration;
	MC_MoveVelocity_0.Deceleration  := Deceleration;
	MC_MoveVelocity_0.Axis := AxisREF;
	MC_MoveVelocity_0();
	(************************** MC_STOP *****************************)
	MC_Stop_0.Axis := AxisREF;
	MC_Stop_0();
	(***************************MC_HALT******************************)
	MC_Halt_0.Axis := AxisREF;
	MC_Halt_0();
	(************************** MC_RESET ****************************)
	MC_Reset_0.Axis := AxisREF;
	MC_Reset_0();
END_FUNCTION_BLOCK
```
